FUNCTION_BLOCK "fbArchiveEquipExhaust"
{ S7_Optimized_Access := 'TRUE' }
VERSION : 0.8
   VAR
      equipmentExhaust { ExternalWritable := 'False'} : Array[1..3] of "tEquipment";
   END_VAR

   VAR_TEMP
      tempInt : Int;
   END_VAR


BEGIN
END_FUNCTION_BLOCK

